paintParameter[1]={vel1 3.00000,velRot1 400.000,velSweep 0.00700000,vel2 3.00000,velRot2 400.000,tPaint1 1.20000,tHex 1.50000,tPaint2 1.50000,tPaint3 1.40000,incrementoZ 95.0000}
paintParameter[2]={vel1 3.00000,velRot1 400.000,velSweep 0.0170000,vel2 3.00000,velRot2 400.000,tPaint1 0.800000,tHex 1.50000,tPaint2 1.50000,tPaint3 1.20000,incrementoZ 95.0000}
paintParameter[3]={vel1 3.00000,velRot1 400.000,velSweep 0.00700000,vel2 3.00000,velRot2 400.000,tPaint1 1.20000,tHex 1.50000,tPaint2 1.50000,tPaint3 1.40000,incrementoZ 95.0000}
paintParameter[4]={vel1 3.00000,velRot1 400.000,velSweep 0.0150000,vel2 3.00000,velRot2 1.00000,tPaint1 2.50000,tHex 1.50000,tPaint2 1.50000,tPaint3 2.50000,incrementoZ 90.0000}
paintParameter[5]={vel1 3.00000,velRot1 400.000,velSweep 0.00700000,vel2 3.00000,velRot2 400.000,tPaint1 1.20000,tHex 1.50000,tPaint2 1.50000,tPaint3 1.40000,incrementoZ 95.0000}
paintParameter[6]={vel1 3.00000,velRot1 400.000,velSweep 0.0200000,vel2 3.00000,velRot2 400.000,tPaint1 0.900000,tHex 1.50000,tPaint2 1.50000,tPaint3 0.900000,incrementoZ 95.0000}
paintParameter[7]={vel1 3.00000,velRot1 400.000,velSweep 0.00700000,vel2 3.00000,velRot2 400.000,tPaint1 1.20000,tHex 1.50000,tPaint2 1.50000,tPaint3 1.40000,incrementoZ 95.0000}
paintParameter[8]={vel1 3.00000,velRot1 400.000,velSweep 0.00700000,vel2 3.00000,velRot2 400.000,tPaint1 1.20000,tHex 1.50000,tPaint2 1.50000,tPaint3 1.40000,incrementoZ 100.000}
paintParameter[9]={vel1 3.00000,velRot1 400.000,velSweep 0.0170000,vel2 3.00000,velRot2 400.000,tPaint1 1.00000,tHex 1.50000,tPaint2 1.50000,tPaint3 1.30000,incrementoZ 95.0000}
paintParameter[10]={vel1 3.00000,velRot1 400.000,velSweep 0.0120000,vel2 3.00000,velRot2 400.000,tPaint1 1.00000,tHex 1.50000,tPaint2 1.50000,tPaint3 1.50000,incrementoZ 95.0000}
paintParameter[11]={vel1 3.00000,velRot1 400.000,velSweep 0.00700000,vel2 3.00000,velRot2 400.000,tPaint1 1.20000,tHex 1.50000,tPaint2 1.50000,tPaint3 1.40000,incrementoZ 95.0000}
paintParameter[12]={vel1 3.00000,velRot1 400.000,velSweep 0.00700000,vel2 3.00000,velRot2 400.000,tPaint1 1.20000,tHex 1.50000,tPaint2 1.50000,tPaint3 1.40000,incrementoZ 95.0000}
paintParameter[13]={vel1 3.00000,velRot1 400.000,velSweep 0.00700000,vel2 3.00000,velRot2 400.000,tPaint1 1.20000,tHex 1.50000,tPaint2 1.50000,tPaint3 1.40000,incrementoZ 95.0000}
paintParameter[14]={vel1 3.00000,velRot1 400.000,velSweep 0.00700000,vel2 3.00000,velRot2 400.000,tPaint1 1.20000,tHex 1.50000,tPaint2 1.50000,tPaint3 1.40000,incrementoZ 95.0000}
paintParameter[15]={vel1 3.00000,velRot1 400.000,velSweep 0.0180000,vel2 3.00000,velRot2 400.000,tPaint1 0.200000,tHex 1.50000,tPaint2 1.50000,tPaint3 2.00000,incrementoZ 0.0}
paintParameter[16]={vel1 3.00000,velRot1 400.000,velSweep 0.00700000,vel2 3.00000,velRot2 400.000,tPaint1 1.20000,tHex 1.50000,tPaint2 1.50000,tPaint3 1.40000,incrementoZ 95.0000}
paintParameter[17]={vel1 3.00000,velRot1 400.000,velSweep 0.00700000,vel2 3.00000,velRot2 400.000,tPaint1 1.20000,tHex 1.50000,tPaint2 1.50000,tPaint3 1.40000,incrementoZ 95.0000}
paintParameter[18]={vel1 3.00000,velRot1 400.000,velSweep 0.0200000,vel2 3.00000,velRot2 400.000,tPaint1 1.20000,tHex 1.50000,tPaint2 1.50000,tPaint3 1.40000,incrementoZ 95.0000}
paintParameter[19]={vel1 3.00000,velRot1 400.000,velSweep 0.00700000,vel2 3.00000,velRot2 400.000,tPaint1 1.20000,tHex 1.50000,tPaint2 1.50000,tPaint3 1.40000,incrementoZ 95.0000}
paintParameter[20]={vel1 3.00000,velRot1 400.000,velSweep 0.00700000,vel2 3.00000,velRot2 400.000,tPaint1 1.20000,tHex 1.50000,tPaint2 1.50000,tPaint3 1.40000,incrementoZ 95.0000}
paintParameter[21]={vel1 3.00000,velRot1 400.000,velSweep 0.00700000,vel2 3.00000,velRot2 400.000,tPaint1 1.20000,tHex 1.50000,tPaint2 1.50000,tPaint3 1.40000,incrementoZ 95.0000}
paintParameter[22]={vel1 3.00000,velRot1 400.000,velSweep 0.00700000,vel2 3.00000,velRot2 400.000,tPaint1 1.20000,tHex 1.50000,tPaint2 1.50000,tPaint3 1.40000,incrementoZ 95.0000}
paintParameter[23]={vel1 3.00000,velRot1 400.000,velSweep 0.00700000,vel2 3.00000,velRot2 400.000,tPaint1 1.20000,tHex 1.50000,tPaint2 1.50000,tPaint3 1.40000,incrementoZ 95.0000}
paintParameter[24]={vel1 3.00000,velRot1 400.000,velSweep 0.00700000,vel2 3.00000,velRot2 400.000,tPaint1 1.20000,tHex 1.50000,tPaint2 1.50000,tPaint3 1.40000,incrementoZ 95.0000}
paintParameter[25]={vel1 3.00000,velRot1 400.000,velSweep 0.00700000,vel2 3.00000,velRot2 400.000,tPaint1 1.20000,tHex 1.50000,tPaint2 1.50000,tPaint3 1.40000,incrementoZ 95.0000}
paintParameter[26]={vel1 3.00000,velRot1 400.000,velSweep 0.00700000,vel2 3.00000,velRot2 400.000,tPaint1 1.20000,tHex 1.50000,tPaint2 1.50000,tPaint3 1.40000,incrementoZ 95.0000}
paintParameter[27]={vel1 3.00000,velRot1 400.000,velSweep 0.00700000,vel2 3.00000,velRot2 400.000,tPaint1 1.20000,tHex 1.50000,tPaint2 1.50000,tPaint3 1.40000,incrementoZ 95.0000}
paintParameter[28]={vel1 3.00000,velRot1 400.000,velSweep 0.00700000,vel2 3.00000,velRot2 400.000,tPaint1 1.20000,tHex 1.50000,tPaint2 1.50000,tPaint3 1.40000,incrementoZ 95.0000}
paintParameter[29]={vel1 3.00000,velRot1 400.000,velSweep 0.00700000,vel2 3.00000,velRot2 400.000,tPaint1 1.20000,tHex 1.50000,tPaint2 1.50000,tPaint3 1.40000,incrementoZ 95.0000}
paintParameter[30]={vel1 3.00000,velRot1 400.000,velSweep 0.00700000,vel2 3.00000,velRot2 400.000,tPaint1 1.20000,tHex 1.50000,tPaint2 1.50000,tPaint3 1.40000,incrementoZ 95.0000}
paintParameter[31]={vel1 3.00000,velRot1 400.000,velSweep 0.00700000,vel2 3.00000,velRot2 400.000,tPaint1 1.20000,tHex 1.50000,tPaint2 1.50000,tPaint3 1.40000,incrementoZ 95.0000}
paintParameter[32]={vel1 3.00000,velRot1 400.000,velSweep 0.00700000,vel2 3.00000,velRot2 400.000,tPaint1 1.20000,tHex 1.50000,tPaint2 1.50000,tPaint3 1.40000,incrementoZ 95.0000}
paintParameter[33]={vel1 3.00000,velRot1 400.000,velSweep 0.00700000,vel2 3.00000,velRot2 400.000,tPaint1 1.20000,tHex 1.50000,tPaint2 1.50000,tPaint3 1.40000,incrementoZ 95.0000}
paintParameter[34]={vel1 3.00000,velRot1 400.000,velSweep 0.00700000,vel2 3.00000,velRot2 400.000,tPaint1 1.20000,tHex 1.50000,tPaint2 1.50000,tPaint3 1.40000,incrementoZ 95.0000}
paintParameter[35]={vel1 3.00000,velRot1 400.000,velSweep 0.00700000,vel2 3.00000,velRot2 400.000,tPaint1 1.20000,tHex 1.50000,tPaint2 1.50000,tPaint3 1.40000,incrementoZ 95.0000}
paintParameter[36]={vel1 3.00000,velRot1 400.000,velSweep 0.00700000,vel2 3.00000,velRot2 400.000,tPaint1 1.20000,tHex 1.50000,tPaint2 1.50000,tPaint3 1.40000,incrementoZ 95.0000}
paintParameter[37]={vel1 3.00000,velRot1 400.000,velSweep 0.00700000,vel2 3.00000,velRot2 400.000,tPaint1 1.20000,tHex 1.50000,tPaint2 1.50000,tPaint3 1.40000,incrementoZ 95.0000}
paintParameter[38]={vel1 3.00000,velRot1 400.000,velSweep 0.00700000,vel2 3.00000,velRot2 400.000,tPaint1 1.20000,tHex 1.50000,tPaint2 1.50000,tPaint3 1.40000,incrementoZ 95.0000}
paintParameter[39]={vel1 3.00000,velRot1 400.000,velSweep 0.00700000,vel2 3.00000,velRot2 400.000,tPaint1 1.20000,tHex 1.50000,tPaint2 1.50000,tPaint3 1.40000,incrementoZ 95.0000}
paintParameter[40]={vel1 3.00000,velRot1 400.000,velSweep 0.00700000,vel2 3.00000,velRot2 400.000,tPaint1 1.20000,tHex 1.50000,tPaint2 1.50000,tPaint3 1.40000,incrementoZ 95.0000}
paintParameter[41]={vel1 3.00000,velRot1 400.000,velSweep 0.00700000,vel2 3.00000,velRot2 400.000,tPaint1 1.20000,tHex 1.50000,tPaint2 1.50000,tPaint3 1.40000,incrementoZ 95.0000}
paintParameter[42]={vel1 3.00000,velRot1 400.000,velSweep 0.00700000,vel2 3.00000,velRot2 400.000,tPaint1 1.20000,tHex 1.50000,tPaint2 1.50000,tPaint3 1.40000,incrementoZ 95.0000}
paintParameter[43]={vel1 3.00000,velRot1 400.000,velSweep 0.00700000,vel2 3.00000,velRot2 400.000,tPaint1 1.20000,tHex 1.50000,tPaint2 1.50000,tPaint3 1.40000,incrementoZ 95.0000}
paintParameter[44]={vel1 3.00000,velRot1 400.000,velSweep 0.00700000,vel2 3.00000,velRot2 400.000,tPaint1 1.20000,tHex 1.50000,tPaint2 1.50000,tPaint3 1.40000,incrementoZ 95.0000}
paintParameter[45]={vel1 3.00000,velRot1 400.000,velSweep 0.00700000,vel2 3.00000,velRot2 400.000,tPaint1 1.20000,tHex 1.50000,tPaint2 1.50000,tPaint3 1.40000,incrementoZ 95.0000}
paintParameter[46]={vel1 3.00000,velRot1 400.000,velSweep 0.00700000,vel2 3.00000,velRot2 400.000,tPaint1 1.20000,tHex 1.50000,tPaint2 1.50000,tPaint3 1.40000,incrementoZ 95.0000}
paintParameter[47]={vel1 3.00000,velRot1 400.000,velSweep 0.00700000,vel2 3.00000,velRot2 400.000,tPaint1 1.20000,tHex 1.50000,tPaint2 1.50000,tPaint3 1.40000,incrementoZ 95.0000}
paintParameter[48]={vel1 3.00000,velRot1 400.000,velSweep 0.00700000,vel2 3.00000,velRot2 400.000,tPaint1 1.20000,tHex 1.50000,tPaint2 1.50000,tPaint3 1.40000,incrementoZ 95.0000}
paintParameter[49]={vel1 3.00000,velRot1 400.000,velSweep 0.00700000,vel2 3.00000,velRot2 400.000,tPaint1 1.20000,tHex 1.50000,tPaint2 1.50000,tPaint3 1.40000,incrementoZ 95.0000}
paintParameter[50]={vel1 3.00000,velRot1 400.000,velSweep 0.00700000,vel2 3.00000,velRot2 400.000,tPaint1 1.20000,tHex 1.50000,tPaint2 1.50000,tPaint3 1.40000,incrementoZ 95.0000}
paintParameter[51]={vel1 3.00000,velRot1 400.000,velSweep 0.00700000,vel2 3.00000,velRot2 400.000,tPaint1 1.20000,tHex 1.50000,tPaint2 1.50000,tPaint3 1.40000,incrementoZ 95.0000}
paintParameter[52]={vel1 3.00000,velRot1 400.000,velSweep 0.00700000,vel2 3.00000,velRot2 400.000,tPaint1 1.20000,tHex 1.50000,tPaint2 1.50000,tPaint3 1.40000,incrementoZ 95.0000}
paintParameter[53]={vel1 3.00000,velRot1 400.000,velSweep 0.00700000,vel2 3.00000,velRot2 400.000,tPaint1 1.20000,tHex 1.50000,tPaint2 1.50000,tPaint3 1.40000,incrementoZ 95.0000}
paintParameter[54]={vel1 3.00000,velRot1 400.000,velSweep 0.00700000,vel2 3.00000,velRot2 400.000,tPaint1 1.20000,tHex 1.50000,tPaint2 1.50000,tPaint3 1.40000,incrementoZ 95.0000}
paintParameter[55]={vel1 3.00000,velRot1 400.000,velSweep 0.00700000,vel2 3.00000,velRot2 400.000,tPaint1 1.20000,tHex 1.50000,tPaint2 1.50000,tPaint3 1.40000,incrementoZ 95.0000}
paintParameter[56]={vel1 3.00000,velRot1 400.000,velSweep 0.00700000,vel2 3.00000,velRot2 400.000,tPaint1 1.20000,tHex 1.50000,tPaint2 1.50000,tPaint3 1.40000,incrementoZ 95.0000}
paintParameter[57]={vel1 3.00000,velRot1 400.000,velSweep 0.00700000,vel2 3.00000,velRot2 400.000,tPaint1 1.20000,tHex 1.50000,tPaint2 1.50000,tPaint3 1.40000,incrementoZ 95.0000}
paintParameter[58]={vel1 3.00000,velRot1 400.000,velSweep 0.00700000,vel2 3.00000,velRot2 400.000,tPaint1 1.20000,tHex 1.50000,tPaint2 1.50000,tPaint3 1.40000,incrementoZ 95.0000}
paintParameter[59]={vel1 3.00000,velRot1 400.000,velSweep 0.00700000,vel2 3.00000,velRot2 400.000,tPaint1 1.20000,tHex 1.50000,tPaint2 1.50000,tPaint3 1.40000,incrementoZ 95.0000}
paintParameter[60]={vel1 3.00000,velRot1 400.000,velSweep 0.00700000,vel2 3.00000,velRot2 400.000,tPaint1 1.20000,tHex 1.50000,tPaint2 1.50000,tPaint3 1.40000,incrementoZ 95.0000}
paintParameter[61]={vel1 3.00000,velRot1 400.000,velSweep 0.00700000,vel2 3.00000,velRot2 400.000,tPaint1 1.20000,tHex 1.50000,tPaint2 1.50000,tPaint3 1.40000,incrementoZ 95.0000}
paintParameter[62]={vel1 3.00000,velRot1 400.000,velSweep 0.00700000,vel2 3.00000,velRot2 400.000,tPaint1 1.20000,tHex 1.50000,tPaint2 1.50000,tPaint3 1.40000,incrementoZ 95.0000}
paintParameter[63]={vel1 3.00000,velRot1 400.000,velSweep 0.00700000,vel2 3.00000,velRot2 400.000,tPaint1 1.20000,tHex 1.50000,tPaint2 1.50000,tPaint3 1.40000,incrementoZ 95.0000}
paintParameter[64]={vel1 3.00000,velRot1 400.000,velSweep 0.00700000,vel2 3.00000,velRot2 400.000,tPaint1 1.20000,tHex 1.50000,tPaint2 1.50000,tPaint3 1.40000,incrementoZ 95.0000}
paintParameter[65]={vel1 3.00000,velRot1 400.000,velSweep 0.00700000,vel2 3.00000,velRot2 400.000,tPaint1 1.20000,tHex 1.50000,tPaint2 1.50000,tPaint3 1.40000,incrementoZ 95.0000}
paintParameter[66]={vel1 3.00000,velRot1 400.000,velSweep 0.00700000,vel2 3.00000,velRot2 400.000,tPaint1 1.20000,tHex 1.50000,tPaint2 1.50000,tPaint3 1.40000,incrementoZ 95.0000}
paintParameter[67]={vel1 3.00000,velRot1 400.000,velSweep 0.00700000,vel2 3.00000,velRot2 400.000,tPaint1 1.20000,tHex 1.50000,tPaint2 1.50000,tPaint3 1.40000,incrementoZ 95.0000}
paintParameter[68]={vel1 3.00000,velRot1 400.000,velSweep 0.00700000,vel2 3.00000,velRot2 400.000,tPaint1 1.20000,tHex 1.50000,tPaint2 1.50000,tPaint3 1.40000,incrementoZ 95.0000}
paintParameter[69]={vel1 3.00000,velRot1 400.000,velSweep 0.00700000,vel2 3.00000,velRot2 400.000,tPaint1 1.20000,tHex 1.50000,tPaint2 1.50000,tPaint3 1.40000,incrementoZ 95.0000}
paintParameter[70]={vel1 3.00000,velRot1 400.000,velSweep 0.00700000,vel2 3.00000,velRot2 400.000,tPaint1 1.20000,tHex 1.50000,tPaint2 1.50000,tPaint3 1.40000,incrementoZ 95.0000}
paintParameter[71]={vel1 3.00000,velRot1 400.000,velSweep 0.00700000,vel2 3.00000,velRot2 400.000,tPaint1 1.20000,tHex 1.50000,tPaint2 1.50000,tPaint3 1.40000,incrementoZ 95.0000}
paintParameter[72]={vel1 3.00000,velRot1 400.000,velSweep 0.00700000,vel2 3.00000,velRot2 400.000,tPaint1 1.20000,tHex 1.50000,tPaint2 1.50000,tPaint3 1.40000,incrementoZ 95.0000}
paintParameter[73]={vel1 3.00000,velRot1 400.000,velSweep 0.00700000,vel2 3.00000,velRot2 400.000,tPaint1 1.20000,tHex 1.50000,tPaint2 1.50000,tPaint3 1.40000,incrementoZ 95.0000}
paintParameter[74]={vel1 3.00000,velRot1 400.000,velSweep 0.00700000,vel2 3.00000,velRot2 400.000,tPaint1 1.20000,tHex 1.50000,tPaint2 1.50000,tPaint3 1.40000,incrementoZ 95.0000}
paintParameter[75]={vel1 3.00000,velRot1 400.000,velSweep 0.00700000,vel2 3.00000,velRot2 400.000,tPaint1 1.20000,tHex 1.50000,tPaint2 1.50000,tPaint3 1.40000,incrementoZ 95.0000}
paintParameter[76]={vel1 3.00000,velRot1 400.000,velSweep 0.00700000,vel2 3.00000,velRot2 400.000,tPaint1 1.20000,tHex 1.50000,tPaint2 1.50000,tPaint3 1.40000,incrementoZ 95.0000}
paintParameter[77]={vel1 3.00000,velRot1 400.000,velSweep 0.00700000,vel2 3.00000,velRot2 400.000,tPaint1 1.20000,tHex 1.50000,tPaint2 1.50000,tPaint3 1.40000,incrementoZ 95.0000}
paintParameter[78]={vel1 3.00000,velRot1 400.000,velSweep 0.00700000,vel2 3.00000,velRot2 400.000,tPaint1 1.20000,tHex 1.50000,tPaint2 1.50000,tPaint3 1.40000,incrementoZ 95.0000}
paintParameter[79]={vel1 3.00000,velRot1 400.000,velSweep 0.00700000,vel2 3.00000,velRot2 400.000,tPaint1 1.20000,tHex 1.50000,tPaint2 1.50000,tPaint3 1.40000,incrementoZ 95.0000}
paintParameter[80]={vel1 3.00000,velRot1 400.000,velSweep 0.00700000,vel2 3.00000,velRot2 400.000,tPaint1 1.20000,tHex 1.50000,tPaint2 1.50000,tPaint3 1.40000,incrementoZ 95.0000}
paintParameter[81]={vel1 3.00000,velRot1 400.000,velSweep 0.00700000,vel2 3.00000,velRot2 400.000,tPaint1 1.20000,tHex 1.50000,tPaint2 1.50000,tPaint3 1.40000,incrementoZ 95.0000}
paintParameter[82]={vel1 3.00000,velRot1 400.000,velSweep 0.00700000,vel2 3.00000,velRot2 400.000,tPaint1 1.20000,tHex 1.50000,tPaint2 1.50000,tPaint3 1.40000,incrementoZ 95.0000}
paintParameter[83]={vel1 3.00000,velRot1 400.000,velSweep 0.00700000,vel2 3.00000,velRot2 400.000,tPaint1 1.20000,tHex 1.50000,tPaint2 1.50000,tPaint3 1.40000,incrementoZ 95.0000}
paintParameter[84]={vel1 3.00000,velRot1 400.000,velSweep 0.00700000,vel2 3.00000,velRot2 400.000,tPaint1 1.20000,tHex 1.50000,tPaint2 1.50000,tPaint3 1.40000,incrementoZ 95.0000}
paintParameter[85]={vel1 3.00000,velRot1 400.000,velSweep 0.00700000,vel2 3.00000,velRot2 400.000,tPaint1 1.20000,tHex 1.50000,tPaint2 1.50000,tPaint3 1.40000,incrementoZ 95.0000}
paintParameter[86]={vel1 3.00000,velRot1 400.000,velSweep 0.00700000,vel2 3.00000,velRot2 400.000,tPaint1 1.20000,tHex 1.50000,tPaint2 1.50000,tPaint3 1.40000,incrementoZ 95.0000}
paintParameter[87]={vel1 3.00000,velRot1 400.000,velSweep 0.00700000,vel2 3.00000,velRot2 400.000,tPaint1 1.20000,tHex 1.50000,tPaint2 1.50000,tPaint3 1.40000,incrementoZ 95.0000}
paintParameter[88]={vel1 3.00000,velRot1 400.000,velSweep 0.00700000,vel2 3.00000,velRot2 400.000,tPaint1 1.20000,tHex 1.50000,tPaint2 1.50000,tPaint3 1.40000,incrementoZ 95.0000}
paintParameter[89]={vel1 3.00000,velRot1 400.000,velSweep 0.00700000,vel2 3.00000,velRot2 400.000,tPaint1 1.20000,tHex 1.50000,tPaint2 1.50000,tPaint3 1.40000,incrementoZ 95.0000}
paintParameter[90]={vel1 3.00000,velRot1 400.000,velSweep 0.00700000,vel2 3.00000,velRot2 400.000,tPaint1 1.20000,tHex 1.50000,tPaint2 1.50000,tPaint3 1.40000,incrementoZ 95.0000}
paintParameter[91]={vel1 3.00000,velRot1 400.000,velSweep 0.00700000,vel2 3.00000,velRot2 400.000,tPaint1 1.20000,tHex 1.50000,tPaint2 1.50000,tPaint3 1.40000,incrementoZ 95.0000}
paintParameter[92]={vel1 3.00000,velRot1 400.000,velSweep 0.00700000,vel2 3.00000,velRot2 400.000,tPaint1 1.20000,tHex 1.50000,tPaint2 1.50000,tPaint3 1.40000,incrementoZ 95.0000}
paintParameter[93]={vel1 3.00000,velRot1 400.000,velSweep 0.00700000,vel2 3.00000,velRot2 400.000,tPaint1 1.20000,tHex 1.50000,tPaint2 1.50000,tPaint3 1.40000,incrementoZ 95.0000}
paintParameter[94]={vel1 3.00000,velRot1 400.000,velSweep 0.00700000,vel2 3.00000,velRot2 400.000,tPaint1 1.20000,tHex 1.50000,tPaint2 1.50000,tPaint3 1.40000,incrementoZ 95.0000}
paintParameter[95]={vel1 3.00000,velRot1 400.000,velSweep 0.00700000,vel2 3.00000,velRot2 400.000,tPaint1 1.20000,tHex 1.50000,tPaint2 1.50000,tPaint3 1.40000,incrementoZ 95.0000}
paintParameter[96]={vel1 3.00000,velRot1 400.000,velSweep 0.00700000,vel2 3.00000,velRot2 400.000,tPaint1 1.20000,tHex 1.50000,tPaint2 1.50000,tPaint3 1.40000,incrementoZ 95.0000}
paintParameter[97]={vel1 3.00000,velRot1 400.000,velSweep 0.00700000,vel2 3.00000,velRot2 400.000,tPaint1 1.20000,tHex 1.50000,tPaint2 1.50000,tPaint3 1.40000,incrementoZ 95.0000}
paintParameter[98]={vel1 3.00000,velRot1 400.000,velSweep 0.00700000,vel2 3.00000,velRot2 400.000,tPaint1 1.20000,tHex 1.50000,tPaint2 1.50000,tPaint3 1.40000,incrementoZ 95.0000}
paintParameter[99]={vel1 3.00000,velRot1 400.000,velSweep 0.00700000,vel2 3.00000,velRot2 400.000,tPaint1 1.20000,tHex 1.50000,tPaint2 1.50000,tPaint3 1.40000,incrementoZ 95.0000}
paintParameter[100]={vel1 3.00000,velRot1 400.000,velSweep 0.00700000,vel2 3.00000,velRot2 400.000,tPaint1 1.20000,tHex 1.50000,tPaint2 1.50000,tPaint3 1.40000,incrementoZ 95.0000}
paintParameter[101]={vel1 3.00000,velRot1 400.000,velSweep 0.00700000,vel2 3.00000,velRot2 400.000,tPaint1 1.20000,tHex 1.50000,tPaint2 1.50000,tPaint3 1.40000,incrementoZ 95.0000}
paintParameter[102]={vel1 3.00000,velRot1 400.000,velSweep 0.00700000,vel2 3.00000,velRot2 400.000,tPaint1 1.20000,tHex 1.50000,tPaint2 1.50000,tPaint3 1.40000,incrementoZ 95.0000}
paintParameter[103]={vel1 3.00000,velRot1 400.000,velSweep 0.00700000,vel2 3.00000,velRot2 400.000,tPaint1 1.20000,tHex 1.50000,tPaint2 1.50000,tPaint3 1.40000,incrementoZ 95.0000}
paintParameter[104]={vel1 3.00000,velRot1 400.000,velSweep 0.00700000,vel2 3.00000,velRot2 400.000,tPaint1 1.20000,tHex 1.50000,tPaint2 1.50000,tPaint3 1.40000,incrementoZ 95.0000}
paintParameter[105]={vel1 3.00000,velRot1 400.000,velSweep 0.00700000,vel2 3.00000,velRot2 400.000,tPaint1 1.20000,tHex 1.50000,tPaint2 1.50000,tPaint3 1.40000,incrementoZ 95.0000}
paintParameter[106]={vel1 3.00000,velRot1 400.000,velSweep 0.00700000,vel2 3.00000,velRot2 400.000,tPaint1 1.20000,tHex 1.50000,tPaint2 1.50000,tPaint3 1.40000,incrementoZ 95.0000}
paintParameter[107]={vel1 3.00000,velRot1 400.000,velSweep 0.00700000,vel2 3.00000,velRot2 400.000,tPaint1 1.20000,tHex 1.50000,tPaint2 1.50000,tPaint3 1.40000,incrementoZ 95.0000}
paintParameter[108]={vel1 3.00000,velRot1 400.000,velSweep 0.00700000,vel2 3.00000,velRot2 400.000,tPaint1 1.20000,tHex 1.50000,tPaint2 1.50000,tPaint3 1.40000,incrementoZ 95.0000}
paintParameter[109]={vel1 3.00000,velRot1 400.000,velSweep 0.00700000,vel2 3.00000,velRot2 400.000,tPaint1 1.20000,tHex 1.50000,tPaint2 1.50000,tPaint3 1.40000,incrementoZ 95.0000}
paintParameter[110]={vel1 3.00000,velRot1 400.000,velSweep 0.00700000,vel2 3.00000,velRot2 400.000,tPaint1 1.20000,tHex 1.50000,tPaint2 1.50000,tPaint3 1.40000,incrementoZ 95.0000}
paintParameter[111]={vel1 3.00000,velRot1 400.000,velSweep 0.00700000,vel2 3.00000,velRot2 400.000,tPaint1 1.20000,tHex 1.50000,tPaint2 1.50000,tPaint3 1.40000,incrementoZ 95.0000}
paintParameter[112]={vel1 3.00000,velRot1 400.000,velSweep 0.00700000,vel2 3.00000,velRot2 400.000,tPaint1 1.20000,tHex 1.50000,tPaint2 1.50000,tPaint3 1.40000,incrementoZ 95.0000}
paintParameter[113]={vel1 3.00000,velRot1 400.000,velSweep 0.00700000,vel2 3.00000,velRot2 400.000,tPaint1 1.20000,tHex 1.50000,tPaint2 1.50000,tPaint3 1.40000,incrementoZ 95.0000}
paintParameter[114]={vel1 3.00000,velRot1 400.000,velSweep 0.00700000,vel2 3.00000,velRot2 400.000,tPaint1 1.20000,tHex 1.50000,tPaint2 1.50000,tPaint3 1.40000,incrementoZ 95.0000}
paintParameter[115]={vel1 3.00000,velRot1 400.000,velSweep 0.00700000,vel2 3.00000,velRot2 400.000,tPaint1 1.20000,tHex 1.50000,tPaint2 1.50000,tPaint3 1.40000,incrementoZ 95.0000}
paintParameter[116]={vel1 3.00000,velRot1 400.000,velSweep 0.00700000,vel2 3.00000,velRot2 400.000,tPaint1 1.20000,tHex 1.50000,tPaint2 1.50000,tPaint3 1.40000,incrementoZ 95.0000}
paintParameter[117]={vel1 3.00000,velRot1 400.000,velSweep 0.00700000,vel2 3.00000,velRot2 400.000,tPaint1 1.20000,tHex 1.50000,tPaint2 1.50000,tPaint3 1.40000,incrementoZ 95.0000}
paintParameter[118]={vel1 3.00000,velRot1 400.000,velSweep 0.00700000,vel2 3.00000,velRot2 400.000,tPaint1 1.20000,tHex 1.50000,tPaint2 1.50000,tPaint3 1.40000,incrementoZ 95.0000}
paintParameter[119]={vel1 3.00000,velRot1 400.000,velSweep 0.00700000,vel2 3.00000,velRot2 400.000,tPaint1 1.20000,tHex 1.50000,tPaint2 1.50000,tPaint3 1.40000,incrementoZ 95.0000}
paintParameter[120]={vel1 3.00000,velRot1 400.000,velSweep 0.00700000,vel2 3.00000,velRot2 400.000,tPaint1 1.20000,tHex 1.50000,tPaint2 1.50000,tPaint3 1.40000,incrementoZ 95.0000}
paintParameter[121]={vel1 3.00000,velRot1 400.000,velSweep 0.00700000,vel2 3.00000,velRot2 400.000,tPaint1 1.20000,tHex 1.50000,tPaint2 1.50000,tPaint3 1.40000,incrementoZ 95.0000}
paintParameter[122]={vel1 3.00000,velRot1 400.000,velSweep 0.00700000,vel2 3.00000,velRot2 400.000,tPaint1 1.20000,tHex 1.50000,tPaint2 1.50000,tPaint3 1.40000,incrementoZ 95.0000}
paintParameter[123]={vel1 3.00000,velRot1 400.000,velSweep 0.00700000,vel2 3.00000,velRot2 400.000,tPaint1 1.20000,tHex 1.50000,tPaint2 1.50000,tPaint3 1.40000,incrementoZ 95.0000}
paintParameter[124]={vel1 3.00000,velRot1 400.000,velSweep 0.00700000,vel2 3.00000,velRot2 400.000,tPaint1 1.20000,tHex 1.50000,tPaint2 1.50000,tPaint3 1.40000,incrementoZ 95.0000}
paintParameter[125]={vel1 3.00000,velRot1 400.000,velSweep 0.00700000,vel2 3.00000,velRot2 400.000,tPaint1 1.20000,tHex 1.50000,tPaint2 1.50000,tPaint3 1.40000,incrementoZ 95.0000}
paintParameter[126]={vel1 3.00000,velRot1 400.000,velSweep 0.00700000,vel2 3.00000,velRot2 400.000,tPaint1 1.20000,tHex 1.50000,tPaint2 1.50000,tPaint3 1.40000,incrementoZ 95.0000}
paintParameter[127]={vel1 3.00000,velRot1 400.000,velSweep 0.00700000,vel2 3.00000,velRot2 400.000,tPaint1 1.20000,tHex 1.50000,tPaint2 1.50000,tPaint3 1.40000,incrementoZ 95.0000}
paintParameter[128]={vel1 3.00000,velRot1 400.000,velSweep 0.00700000,vel2 3.00000,velRot2 400.000,tPaint1 1.20000,tHex 1.50000,tPaint2 1.50000,tPaint3 1.40000,incrementoZ 95.0000}

;==================================
; Vars unicas
;==================================
DECL CONST POS $NULLPOS={X 0.0,Y 0.0,Z 0.0,A 0.0,B 0.0,C 0.0,S 0,T 0}
DECL INT primerBitPresencia=272
DECL INT primerBitMemoria=172
DECL BOOL posicionesTest[8]
posicionesTest[1]=FALSE
posicionesTest[2]=FALSE
posicionesTest[3]=FALSE
posicionesTest[4]=FALSE
posicionesTest[5]=FALSE
posicionesTest[6]=FALSE
posicionesTest[7]=FALSE
posicionesTest[8]=FALSE

;DECL BOOL memoriasPresencia[4,2]
;memoriasPresencia[1,1] = False
;memoriasPresencia[2,1] = False
;memoriasPresencia[3,1] = False
;memoriasPresencia[4,1] = False
;memoriasPresencia[1,2] = False
;memoriasPresencia[2,2] = False
;memoriasPresencia[3,2] = False
;memoriasPresencia[4,2] = False


;==================================
; Recetas
;==================================

DECL CHAR RECIPE_NAME[128,24]
RECIPE_NAME[1,]="TR47H90L210"
RECIPE_NAME[2,]="ER60H60L550"
RECIPE_NAME[3,]="ER39H39L1000"


DECL PIECE_TYPE PIECE_TYPE_AR[128]
PIECE_TYPE_AR[1]=#Tornillo
PIECE_TYPE_AR[2]=#Esparrago
PIECE_TYPE_AR[3]=#Esparrago
PIECE_TYPE_AR[20]=#Esparrago


DECL FRAME RECIPE_TCP[128]
RECIPE_TCP[1]={X 413.950287,Y 670.396179,Z 143.821548,A 0.0,B -90.0000,C 0.0}
RECIPE_TCP[2]={X 413.950287,Y 670.396179,Z 143.821548,A 0.0,B -90.0000,C 0.0}
RECIPE_TCP[3]={X 413.950287,Y 670.396179,Z 143.821548,A 0.0,B -90.0000,C 0.0}
RECIPE_TCP[20]={X 413.950287,Y 670.396179,Z 143.821548,A 0.0,B -90.0000,C 0.0}

DECL RECIPE_TYPE $RECIPE={lTotal 350.000,lOffsetCBP 110.000,lOffsetCIND 250.000,lHexagono 0.0,diametroHexagono 0.0,diametroRosca 42.0000,recipeNum 15,PiO {X 0.0,Y 0.0,Z 0.0,A 0.0,B 0.0,C 0.0},PlO {X 0.0,Y 0.0,Z 0.0,A 0.0,B 0.0,C 0.0}}


;==================================
; Configuraciones de celda
;==================================
DECL LAYOUT_CONFIG LAYOUT_DATA[16]
LAYOUT_DATA[1]={alphaVBP 90.0000,alphaVIND 60.0000,lIRXOffset 128.000,lIRYOffset 715.000,workAngle 30.0000,maxPiezasIR 4,layoutNum 1}
LAYOUT_DATA[2]={alphaVBP 90.0000,alphaVIND 60.0000,lIRXOffset 128.000,lIRYOffset 715.000,workAngle 30.0000,maxPiezasIR 4,layoutNum 1}

DECL CHAR LAYOUT_NAME[16,24]
LAYOUT_NAME[1,]="Torres Guma"
LAYOUT_NAME[2,]="Erreka Bergara"

DECL FRAME LAYOUT_BASE_PICKBP[16]
LAYOUT_BASE_PICKBP[1]={X -1295.00,Y -2000.00,Z 941.000,A 180.000,B 0.0,C 0.0}

DECL FRAME LAYOUT_BASE_LASERETCP[16]
LAYOUT_BASE_LASERETCP[1]={X 1280.00,Y 530.000,Z 725.000,A 0.0,B -5.00000,C 0.0}

DECL FRAME LAYOUT_BASE_PLACEIR[16]
LAYOUT_BASE_PLACEIR[1]={X 186.682709,Y -2099.32446,Z 768.276062,A -90.0000,B 0.0,C 0.0}

DECL LAYOUT_CONFIG $LAYOUT={alphaVBP 120.000,alphaVIND 60.0000,lIRXOffset 128.000,lIRYOffset 715.000,workAngle 30.0000,maxPiezasIR 4,layoutNum 1}





;ENDFOLD


;ENDFOLD

;ENDFOLD (USER GLOBALS)
;ENDFOLD


;==================================
; Userdefined Externals
;==================================

;==================================
; Userdefined Variables
;==================================

;ENDFOLD (USER GLOBALS)
ENDDAT
